PROGRAM Hardware_3510
VAR
    // Servos *********************************************************************
	fbX_Achse										: FB_Achse_NC_PTP_Beckhoff_V2;  

    // Frequenzumrichter **********************************************************
	fbTrans_Schlossseite							: FB_SEW_MOVITRAC_C_CoE;

    // Sensorik *******************************************************************
    fbLangsam          								: FB_Belegt;
    fbStopp         								: FB_Belegt;
    fbLaengsSchlossseite_Ref						: FB_Belegt;

    // Ventile ********************************************************************
    fbLaengsanschl                					: FB_Ventil_V2;
    fbSchienenklemm               					: FB_Ventil_V2;

    // ***** Hilfsmerker***********************************************************
    (*
        Ventile sind über den DUT_Ventil_para vorparametriert
                ueberwachung_vor_aktiv    : BOOL := TRUE;   // 0 = Endlagenüberwachung vor deaktiviert
                ueberwachung_zur_aktiv    : BOOL := TRUE;   // 0 = Endlagenüberwachung zurück deaktiviert
                ausgang_vor_halten        : BOOL := FALSE;  // 1 = Ausgang immer Ein, sonst 0 in Endlage/1 nicht in Endlage
                ausgang_zur_halten        : BOOL := FALSE;  // 1 = Ausgang immer Ein, sonst 0 in Endlage/1 nicht in Endlage
                entprellen_vor_aktiv      : BOOL := TRUE;   // 0 = Endlage sofort überwachen wenn einmal erreicht
                entprellen_zur_aktiv      : BOOL := TRUE;   // 0 = Endlage sofort überwachen wenn einmal erreicht
                ueberwachungszeit_vor     : TIME := T#10S;  // Überwachungszeit in ms (0-30000ms)
                ueberwachungszeit_zur     : TIME := T#10S;  // Überwachungszeit in ms (0-30000ms)
                entprellungszeit_vor      : TIME := T#50MS; // Entprellungszeit in ms (0-10000ms)
                entprellungszeit_zur      : TIME := T#50MS; // Entprellungszeit in ms (0-10000ms)

        falls etwas anderes gewünscht ist, kann man gezielt für das Ventil die Parameter anpassen
        Beispiel:   ***.para.ausgang_vor_halten := TRUE;
                    ***.para.entprellungszeit_vor := T#100MS;
    *)
END_VAR


// Aktionen aufrufen
//_________________________________________________
	A_Sensorik();
	A_Umrichter();
	A_Ventile();
	A_Servo();

ACTION A_Sensorik:
					
// ***** Sensorik entprellen *********************************************************
	//********************************************************************************
fbLangsam						(	in_Sensor:=,
									in_zeit_aus:=T#100MS,
									in_zeit_aus:=T#100MS,
									Q=>);
									
fbStopp							(	in_Sensor:=,
									in_zeit_aus:=T#100MS,
									in_zeit_aus:=T#100MS,
									Q=>);
									
fbLaengsSchlossseite_Ref		(	in_Sensor:=,
									in_zeit_aus:=T#100MS,
									in_zeit_aus:=T#100MS,
									Q=>);
END_ACTION

ACTION A_Servo:
					
// ***** Servoregler *****************************************************************
	//********************************************************************************
								
	GVL_3510.X_Achse_steuern.Reglersperre	:= GVL_3000.bAchsen_Reglersperre;
	GVL_3510.X_Achse_steuern.Freigabe 		:= GVL_3000.bAchsen_Freigabe;
	
	fbX_Achse(
	in_Reglersperre				:= GVL_3510.X_Achse_steuern.Reglersperre, 
	in_Freigabe					:= GVL_3510.X_Achse_steuern.Freigabe,
	in_Reset					:= GVL_Visu_3510.SteuerStatus.reset   
								OR GVL_3000.stoerung_quitt,                      
	in_Hand						:= GVL_Visu_3510.SteuerStatus.hand,              
	in_Auto						:= GVL_Visu_3510.SteuerStatus.auto,                 
	in_Auto_Override			:= GVL_Visu_3000.override,    
	in_Auto_pos					:= , 
	in_max_Velo					:= 100 ,
	in_PosFenster				:= 0.05, 
	in_Ref_pos					:= 0.0, 
	in_HomingOption				:= , 
	in_EndlageRef				:= , 
	in_DirRef					:= , 
	in_PosEa					:= ,                                       
	out_ist_pos					=> GVL_3510.X_Achse_status.ist_pos, 
	out_in_pos					=> GVL_3510.X_Achse_status.in_pos,   
	out_ziel_pos				=> GVL_3510.X_Achse_status.ziel_pos, 
	out_nicht_ref				=> GVL_3510.X_Achse_status.nicht_ref,      
	out_bremse					=> GVL_3510.X_Achse_status.bremse,           
	out_Achs_Status				=> GVL_3510.X_Achse_status.Achs_Status,  
	inout_NC					:= EAs_3510.ea_X_Achse, 
	inout_service				:= GVL_Visu_3510.X_Achse, 
	inout_Ref_start				:= GVL_3510.X_Achse_steuern.Ref_start, 
	inout_Auto_start			:= GVL_3510.X_Achse_steuern.Auto_start, 
	inout_Auto_stop				:= GVL_3510.X_Achse_steuern.Auto_stop);
	
	GVL_Meldungen.Diagnose_3000.Nr_104	:= fbX_Achse.out_Achs_ErrorID;	
	GVL_Meldungen.Meldungen_3000.Nr_104 := fbX_Achse.out_Achs_Error OR fbX_Achse.out_FB_Error OR fbX_Achse.out_Achs_ErrorID <> 0;		
	GVL_Meldungen.Meldungen_3000.Nr_105 := FALSE;
	GVL_Meldungen.Meldungen_3000.Nr_106 := FALSE;
END_ACTION

ACTION A_Umrichter:

// ***** Frequenzumrichter ******************************************************
// ******************************************************************************
				
	GVL_Visu_3510.Trans_Schlossseite	.Para.Speed_Hand		:= 20;
	GVL_Visu_3510.Trans_Schlossseite	.Para.Beschleunigung 	:= 10000;
	GVL_Visu_3510.Trans_Schlossseite	.Para.Verzoegerung 		:= 10000;
	GVL_Visu_3510.Trans_Schlossseite	.Para.Einheit			:= 1;
	GVL_Visu_3510.Trans_Schlossseite	.Para.Kommastelle		:= 1;

	fbTrans_Schlossseite	(	PD_IN	:=EAs_3510.e_Trans_Schlossseite	,
			IN_ReglerSperre			:=not GVL_3000.bAchsen_Reglersperre,
			IN_SteuerStatus			:=GVL_Visu_3510.SteuerStatus,
			IN_Ethercat_Adresse		:=,
			IN_Ethercat_Name		:='',
			IN_QUITTIEREN			:= GVL_3000.stoerung_quitt,
			IN_OVERRIDE				:= GVL_Visu_3000.override,
			PD_OUT					=> EAs_3510.a_Trans_Schlossseite	,
			OUT_Stoerung			=> GVL_Meldungen.Meldungen_3000.Nr_008,
			OUT_Fehlernummer		=> GVL_Meldungen.Diagnose_3000.Nr_008,
			OUT_Status				=> GVL_3510.Trans_Schlossseite_status,
			inout_visu				:= GVL_Visu_3510.Trans_Schlossseite	,
			inout_steuern			:= GVL_3510.Trans_Schlossseite_steuern);
	
			GVL_3510.Trans_Schlossseite_steuern.vor := FALSE;
			GVL_3510.Trans_Schlossseite_steuern.zur := FALSE;
			GVL_3510.Trans_Schlossseite_steuern.speed := 40;
END_ACTION

ACTION A_Ventile:
	
// ***** Ventile *********************************************************************
	//********************************************************************************	
	
	GVL_3510.Laengsanschl.in_freigabe_vor := GVL_3000.bDruckluft_Bereit;
	GVL_3510.Laengsanschl.in_freigabe_zur := GVL_3000.bDruckluft_Bereit;
	GVL_Visu_3510.Laengsanschl.para.ausgang_vor_halten:=TRUE;	
	GVL_Visu_3510.Laengsanschl.para.ausgang_zur_halten:=TRUE;	
	GVL_Visu_3510.Laengsanschl.para.ueberwachung_vor_aktiv:=TRUE;	
	GVL_Visu_3510.Laengsanschl.para.ueberwachung_zur_aktiv:=TRUE;	
	GVL_Visu_3510.Laengsanschl.para.entprellungszeit_vor:=T#50S;	
	GVL_Visu_3510.Laengsanschl.para.entprellungszeit_zur:=T#50MS;	
	fbLaengsanschl (		in_endlage_vor:= ,
							in_endlage_zur:= ,
							in_hand:=GVL_Visu_3510.SteuerStatus.hand,
							in_auto:=GVL_Visu_3510.SteuerStatus.auto,
								in_simu :=GVL_3000.bMode_Sim_Ventile,
							in_quit:=GVL_Visu_3510.SteuerStatus.reset 
							OR GVL_3000.stoerung_quitt,
							out_vor=>,
							out_zur=>,
							out_stoerung_vor=> GVL_Meldungen.Meldungen_3000.Nr_073,
							out_stoerung_zur=> GVL_Meldungen.Meldungen_3000.Nr_074,
							out_stoerung_vorzur=> GVL_Meldungen.Meldungen_3000.Nr_075,
							inout_ansteuerung:=GVL_3510.Laengsanschl ,
							inout_visu:=GVL_Visu_3510.Laengsanschl );
								
	
	GVL_3510.Schienenklemm.in_freigabe_vor := GVL_3000.bDruckluft_Bereit;
	GVL_3510.Schienenklemm.in_freigabe_zur := GVL_3000.bDruckluft_Bereit;
	GVL_Visu_3510.Schienenklemm.para.ausgang_vor_halten:=TRUE;	
	GVL_Visu_3510.Schienenklemm.para.ausgang_zur_halten:=TRUE;	
	GVL_Visu_3510.Schienenklemm.para.ueberwachung_vor_aktiv:=TRUE;	
	GVL_Visu_3510.Schienenklemm.para.ueberwachung_zur_aktiv:=TRUE;	
	GVL_Visu_3510.Schienenklemm.para.entprellungszeit_vor:=T#500MS;	
	GVL_Visu_3510.Schienenklemm.para.entprellungszeit_zur:=T#500MS;	
	fbSchienenklemm(			in_endlage_vor:= EAs_3510.a_FR_3510_Transport_Schlossseite_X_Achse_Laengsanschlag_Schienenklemmung_klemmen, 
								in_endlage_zur:= NOT EAs_3510.a_FR_3510_Transport_Schlossseite_X_Achse_Laengsanschlag_Schienenklemmung_klemmen,
								in_hand:=GVL_Visu_3510.SteuerStatus.hand,
								in_auto:=GVL_Visu_3510.SteuerStatus.auto,
								in_simu :=GVL_3000.bMode_Sim_Ventile,
								in_quit:=GVL_Visu_3510.SteuerStatus.reset 
								OR GVL_3000.stoerung_quitt,
								out_vor=>EAs_3510.a_FR_3510_Transport_Schlossseite_X_Achse_Laengsanschlag_Schienenklemmung_klemmen,
								out_zur=>,
								out_stoerung_vor=> GVL_Meldungen.Meldungen_3000.Nr_088,
								out_stoerung_zur=> GVL_Meldungen.Meldungen_3000.Nr_089,
								out_stoerung_vorzur=> GVL_Meldungen.Meldungen_3000.Nr_090,
								inout_ansteuerung:=GVL_3510.Schienenklemm,
								inout_visu:=GVL_Visu_3510.Schienenklemm);
END_ACTION

END_PROGRAM

(* stored: Version 1.1.0.1
   POU Hardware_3510: Id {e019c143-cdf9-4c7e-96a4-f0c51d8bdf1f}, SpecialFunc None
   Action A_Sensorik: Id {f5beab16-1a04-4437-9743-5acffdc85692}
   Action A_Servo: Id {fff70697-4092-44ed-8a1a-0cfa0e5da105}
   Action A_Umrichter: Id {1e7dffa0-b942-4a9e-be76-2daa42d15cf9}
   Action A_Ventile: Id {c674722c-829e-44a8-828a-026f6fd1b73f} *)
